{attribute 'linkalways'} 
{attribute 'no_explicit_call' := 'This FB is a CLASS and must be accessed using methods or properties'}
{attribute 'enable_dynamic_creation'}
FUNCTION_BLOCK _TcVnPoint3_LREAL EXTENDS AliasDatatypeBase
VAR
	localData : TcVnPoint3_LREAL;
	activeData : REFERENCE TO TcVnPoint3_LREAL REF= localData;
	aliasBaseDatatype : _TcVnVector3_LREAL;
END_VAR

PROPERTY PUBLIC Address : PVOID
GET
Address := ADR(activeData);
END_GET
END_PROPERTY

METHOD PUBLIC ClearReference
VAR_INPUT
END_VAR
activeData REF= localData;
SetBaseDatatypeReference();
END_METHOD

METHOD PUBLIC Clone : I_Datatype
VAR
    pClone : POINTER TO _TcVnPoint3_LREAL;
END_VAR
pClone := __NEW(_TcVnPoint3_LREAL);
Clone := pClone^;
END_METHOD

METHOD FB_init : BOOL
VAR_INPUT
	bInitRetains : BOOL; // if TRUE, the retain variables are initialized (warm start / cold start)
	bInCopyCode : BOOL;  // if TRUE, the instance afterwards gets moved into the copy code (online change)
	//InitialValue : <type>; // if possible, not all values can be initialized
END_VAR
//localData := InitialValue; // if possible, not all values can be initialized
SetBaseDatatypeReference();
AddBaseDatatype(aliasBaseDatatype);
END_METHOD

PROPERTY PUBLIC Identifier : T_MAXSTRING
GET
Identifier := 'TcVnPoint3_LREAL';
END_GET
END_PROPERTY

METHOD PUBLIC MakeReferenceTo
VAR_INPUT
	ReferenceTarget : REFERENCE TO TcVnPoint3_LREAL;
END_VAR
activeData REF= ReferenceTarget;
SetBaseDatatypeReference();
END_METHOD

METHOD PROTECTED SetBaseDatatypeReference
VAR_INPUT
END_VAR
aliasBaseDatatype.MakeReferenceTo(activeData);
END_METHOD

PROPERTY PUBLIC Size : UDINT
GET
Size := SIZEOF(activeData);
END_GET
END_PROPERTY

METHOD TryMakeReferenceTo : BOOL
VAR_INPUT
	Target : I_Datatype;
END_VAR
VAR
	pTargetData : POINTER TO TcVnPoint3_LREAL;
END_VAR
IF NOT IsEquivalentTo(Target) THEN
	RETURN;
END_IF

pTargetData := Target.Address;
activeData REF= pTargetData^;
SetBaseDatatypeReference();
TryMakeReferenceTo := TRUE;
END_METHOD

PROPERTY PUBLIC Value : REFERENCE TO TcVnPoint3_LREAL
GET
Value REF= activeData;
END_GET
END_PROPERTY

END_FUNCTION_BLOCK

(* stored: Version 1.1.0.1, ProductVersion 3.1.4024.13
   POU _TcVnPoint3_LREAL: Id {e2bf02df-9128-0642-38af-aea89987d0ec}, SpecialFunc None
   Folder Core: Id {08703c81-15e0-0783-2f75-304e40d50f2d}
   Folder Protected: Id {944724d7-f130-0bdd-3890-66017f46ac2f}
   Folder Customize: Id {9b2169b8-d9a6-0217-1d45-286f0c52401c}
   Folder Constructor: Id {501876c1-bf7c-0225-1d12-94a6f5cd35bb}
   Property Address: Id {806cff65-7c13-0bd8-30a5-d3a759846243}
   Get Get: Id {4eeed005-93ae-0ae7-0a65-f4d554ca0ed3}
   Method ClearReference: Id {16ab51e7-154b-0763-29c7-1a3d368207f6}
   Method Clone: Id {04acaab2-a5ee-03cf-3861-54906e329ec8}
   Method FB_init: Id {37d03d33-a3f3-05c0-0cfa-ca63de434b72}
   Property Identifier: Id {a98192b7-34f3-077b-21b7-2a78eaf59fd4}
   Get Get: Id {632041ce-c67a-06b4-30ec-e0b8d11205f3}
   Method MakeReferenceTo: Id {ec5f458a-8bad-0388-13af-f380e3883fa5}
   Method SetBaseDatatypeReference: Id {d843fc10-6a41-0bfa-2a4b-73ec4154b4d8}
   Property Size: Id {4b3b2c3c-b01b-0324-1c2d-660a863a2cf3}
   Get Get: Id {f8f06a8d-1360-0cbd-088a-00b562e52cc4}
   Method TryMakeReferenceTo: Id {44507da1-7062-089e-2d9c-1c28e4371812}
   Property Value: Id {93149c3f-d36d-0f0a-2e7f-bb7b5d897156}
   Get Get: Id {ac5e59ce-2795-0f0f-2567-923f5eec19fa} *)
